{attribute 'qualified_only'}
{attribute 'strict'}
{attribute 'to_string'}
TYPE E_3102_Error_status :
(
	no_error := 0,
	error_on	:=1
)UINT;
END_TYPE

(* stored: Version 1.1.0.1, ProductVersion 3.1.4026.17
   DUT E_3102_Error_status: Id {27a4c9b7-6c4a-444b-b309-84151af96d38} *)
